RoboDK station: Example 1.1 - Linear rail & 2 fingers gripper Station.rdk

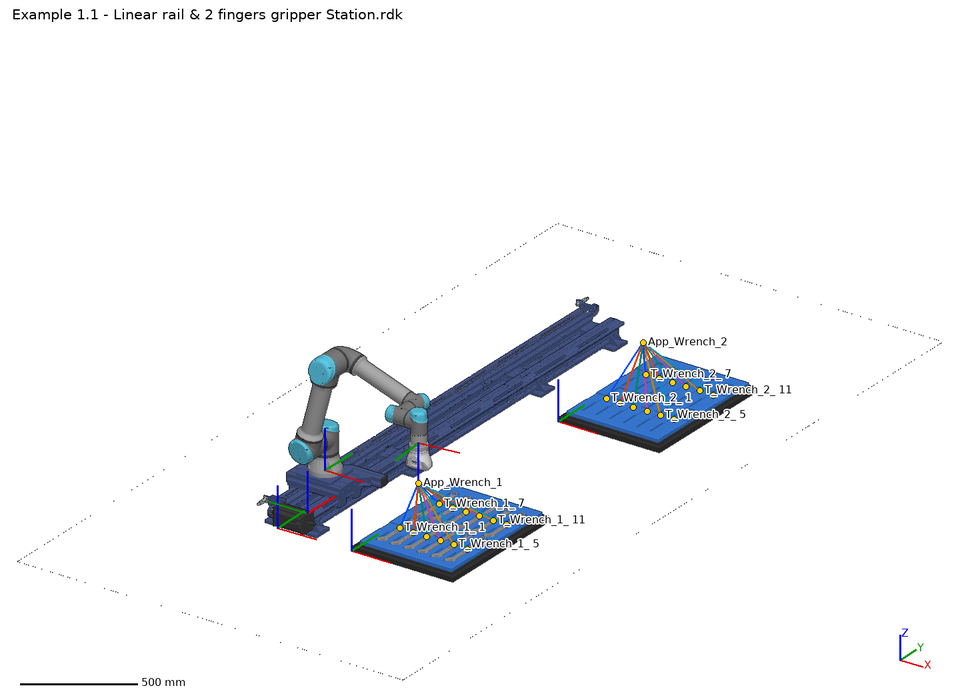
[picture v0: the station drawn from its stored meshes, robots at their saved joint values, targets as dots, program paths as lines]
Station Example 1.1 - 2 fingers gripper Station. Poses are relative to the parent item; angles as X-Y-Z fixed-axis rotations.
  - frame World at (0, 0, 0) mm
    - object Floor at (280, 1100, 0) mm, size 2000 x 4000 x 1 mm, geometry from plane_1m.sld
  - frame Linear Rail Base at (148.81, 12.71, 105) mm, rotated rx 0 ry 0 rz 90 deg
    - robot Linear Rail: 1 axes
        modified DH rows (alpha deg, a mm, theta deg, d mm): 0, 0, 0, 0 linear
        base shift (0, 0, 0) mm, rotated rx 0 ry 90 rz 0 deg
        joint limits [0] to [2100]; home [0]; saved at [150]
      - frame UR5e Base at (100, 85, 80) mm, rotated rx 0 ry 0 rz -90 deg
        - robot UR5e: 6 axes, payload 5 kg, reach 850 mm, repeatability 0.03 mm, weight 18.4 kg
            modified DH rows (alpha deg, a mm, theta deg, d mm): 0, 0, 0, 162.5; 90, 0, 180, 0; 0, 425, 0, 0; 0, 392.25, 0, 133.3; -90, 0, 0, 99.7; 90, 0, 180, 99.6
            joint limits [-360, -360, -360, -360, -360, -360] to [360, 360, 360, 360, 360, 360]; home [0, -90, -90, 0, 90, 0]; saved at [0, -104.57, -94.67, -70.76, 90, -95.16]
          - frame Schunk_Gripper Base at (0, 0, 0) mm
            - robot Schunk_Gripper: 1 axes
                joint limits [0] to [40]; home [40]; saved at [9]
            - target Gripper_Open (joint target) at (-117.49, 235.59, 143.86) mm; joints [40, 0, 0, 0, 0, 0] of Schunk_Gripper
            - target Gripper_Pick (joint target) at (0, 0, 150) mm; joints [9, 0, 0, 0, 0, 0] of Schunk_Gripper
          - tool Shunck_TCP, TCP at (0, 0, 190) mm
    - target Rail_Pos1 (joint target) at (150, 0, 0) mm; joints [150, 0, 0, 0, 0, nan] of Linear Rail
    - target Rail_Pos2 (joint target) at (1814.34, 0, 0) mm; joints [1814.34, 0, 0, 0, 0, 0] of Linear Rail
  - frame Frame Wrench 1 at (386.44, -2.63, 0) mm
    - object Jig at (0, 0, 0) mm, size 525 x 720 x 30 mm, geometry from Jig.step
    - object Wrench Matrix at (25, 25, 10) mm, size 475 x 670 x 40 mm, geometry from Matrix.step
    - target T_Wrench_1_ 1 (Cartesian target) at (100, 215, 50) mm, rotated rx 180 ry 0 rz 0 deg; joints [11.458, -119.591, -136.449, -13.961, 90, -78.542] of UR5e
    - target T_Wrench_1_ 2 (Cartesian target) at (170, 215, 50) mm, rotated rx 180 ry 0 rz 0 deg; joints [9.78, -123.515, -125.176, -21.309, 90, -80.22] of UR5e
    - target T_Wrench_1_ 3 (Cartesian target) at (240, 215, 50) mm, rotated rx 180 ry 0 rz 0 deg; joints [8.536, -128.193, -113.428, -28.378, 90, -81.464] of UR5e
    - target T_Wrench_1_ 4 (Cartesian target) at (310, 215, 50) mm, rotated rx 180 ry 0 rz 0 deg; joints [7.575, -133.539, -100.921, -35.54, 90, -82.425] of UR5e
    - target T_Wrench_1_ 5 (Cartesian target) at (380, 215, 50) mm, rotated rx 180 ry 0 rz 0 deg; joints [6.809, -139.644, -87.232, -43.124, 90, -83.191] of UR5e
    - target T_Wrench_1_ 6 (Cartesian target) at (450, 215, 50) mm, rotated rx 180 ry 0 rz 0 deg; joints [6.185, -146.811, -71.606, -51.583, 90, -83.815] of UR5e
    - target T_Wrench_1_ 7 (Cartesian target) at (100, 505, 50) mm, rotated rx 180 ry 0 rz 0 deg; joints [45.48, -122.94, -126.711, -20.349, 90, -44.52] of UR5e
    - target T_Wrench_1_ 8 (Cartesian target) at (170, 505, 50) mm, rotated rx 180 ry 0 rz 0 deg; joints [40.025, -126.988, -116.359, -26.653, 90, -49.975] of UR5e
    - target T_Wrench_1_ 9 (Cartesian target) at (240, 505, 50) mm, rotated rx 180 ry 0 rz 0 deg; joints [35.662, -131.694, -105.165, -33.141, 90, -54.338] of UR5e
    - target T_Wrench_1_ 10 (Cartesian target) at (310, 505, 50) mm, rotated rx 180 ry 0 rz 0 deg; joints [32.112, -137.097, -92.887, -40.015, 90, -57.888] of UR5e
    - target T_Wrench_1_ 11 (Cartesian target) at (380, 505, 50) mm, rotated rx 180 ry 0 rz 0 deg; joints [29.178, -143.374, -79.056, -47.57, 90, -60.822] of UR5e
    - target T_Wrench_1_ 12 (Cartesian target) at (450, 505, 50) mm, rotated rx 180 ry 0 rz 0 deg; joints [26.718, -150.974, -62.667, -56.359, 90, -63.282] of UR5e
    - target App_Wrench_1 (joint target) at (254.33, 132.05, 339.98) mm, rotated rx 180 ry 0 rz 5.16 deg; joints [0, -104.57, -94.67, -70.76, 90, -95.16] of UR5e
    - object Wrench 11 at (380, 505, 65) mm, size 44.5 x 267.3 x 18.4 mm, geometry from Wrench.step
    - object Wrench 12 at (450, 505, 65) mm, size 44.5 x 267.3 x 18.4 mm, geometry from Wrench.step
    - object Wrench 1 at (100, 215, 65) mm, size 44.5 x 267.3 x 18.4 mm, geometry from Wrench.step
    - object Wrench 2 at (170, 215, 65) mm, size 44.5 x 267.3 x 18.4 mm, geometry from Wrench.step
    - object Wrench 3 at (240, 215, 65) mm, size 44.5 x 267.3 x 18.4 mm, geometry from Wrench.step
    - object Wrench 4 at (310, 215, 65) mm, size 44.5 x 267.3 x 18.4 mm, geometry from Wrench.step
    - object Wrench 5 at (380, 215, 65) mm, size 44.5 x 267.3 x 18.4 mm, geometry from Wrench.step
    - object Wrench 6 at (450, 215, 65) mm, size 44.5 x 267.3 x 18.4 mm, geometry from Wrench.step
    - object Wrench 7 at (100, 505, 65) mm, size 44.5 x 267.3 x 18.4 mm, geometry from Wrench.step
    - object Wrench 8 at (170, 505, 65) mm, size 44.5 x 267.3 x 18.4 mm, geometry from Wrench.step
    - object Wrench 9 at (240, 505, 65) mm, size 44.5 x 267.3 x 18.4 mm, geometry from Wrench.step
    - object Wrench 10 at (310, 505, 65) mm, size 44.5 x 267.3 x 18.4 mm, geometry from Wrench.step
  - frame Frame Wrench 2 at (386.44, 1527.37, 0) mm
    - object Jig at (0, 0, 0) mm, size 525 x 720 x 30 mm, geometry from Jig.step
    - object Wrench Matrix at (25, 25, 10) mm, size 475 x 670 x 40 mm, geometry from Matrix.step
    - target T_Wrench_2_ 1 (Cartesian target) at (100, 215, 50) mm, rotated rx 180 ry 0 rz 0 deg; joints [11.458, -119.591, -136.449, -13.961, 90, -78.542] of UR5e
    - target T_Wrench_2_ 2 (Cartesian target) at (170, 215, 50) mm, rotated rx 180 ry 0 rz 0 deg; joints [9.78, -123.515, -125.176, -21.309, 90, -80.22] of UR5e
    - target T_Wrench_2_ 3 (Cartesian target) at (240, 215, 50) mm, rotated rx 180 ry 0 rz 0 deg; joints [8.536, -128.193, -113.428, -28.378, 90, -81.464] of UR5e
    - target T_Wrench_2_ 4 (Cartesian target) at (310, 215, 50) mm, rotated rx 180 ry 0 rz 0 deg; joints [7.575, -133.539, -100.921, -35.54, 90, -82.425] of UR5e
    - target T_Wrench_2_ 5 (Cartesian target) at (380, 215, 50) mm, rotated rx 180 ry 0 rz 0 deg; joints [6.809, -139.644, -87.232, -43.124, 90, -83.191] of UR5e
    - target T_Wrench_2_ 6 (Cartesian target) at (450, 215, 50) mm, rotated rx 180 ry 0 rz 0 deg; joints [6.185, -146.811, -71.606, -51.583, 90, -83.815] of UR5e
    - target T_Wrench_2_ 7 (Cartesian target) at (100, 505, 50) mm, rotated rx 180 ry 0 rz 0 deg; joints [45.48, -122.94, -126.711, -20.349, 90, -44.52] of UR5e
    - target T_Wrench_2_ 8 (Cartesian target) at (170, 505, 50) mm, rotated rx 180 ry 0 rz 0 deg; joints [40.025, -126.988, -116.359, -26.653, 90, -49.975] of UR5e
    - target T_Wrench_2_ 9 (Cartesian target) at (240, 505, 50) mm, rotated rx 180 ry 0 rz 0 deg; joints [35.662, -131.694, -105.165, -33.141, 90, -54.338] of UR5e
    - target T_Wrench_2_ 10 (Cartesian target) at (310, 505, 50) mm, rotated rx 180 ry 0 rz 0 deg; joints [32.112, -137.097, -92.887, -40.015, 90, -57.888] of UR5e
    - target T_Wrench_2_ 11 (Cartesian target) at (380, 505, 50) mm, rotated rx 180 ry 0 rz 0 deg; joints [29.178, -143.374, -79.056, -47.57, 90, -60.822] of UR5e
    - target T_Wrench_2_ 12 (Cartesian target) at (450, 505, 50) mm, rotated rx 180 ry 0 rz 0 deg; joints [26.718, -150.974, -62.667, -56.359, 90, -63.282] of UR5e
    - target App_Wrench_2 (joint target) at (254.33, 266.39, 339.98) mm, rotated rx 180 ry 0 rz 5.16 deg; joints [0, -104.57, -94.67, -70.76, 90, -95.16] of UR5e
  - program ReplaceObjects (1 instructions, listed below)
  - folder RailPositions
    - program RailPos1 (1 instructions, listed below)
    - program RailPos2 (1 instructions, listed below)
  - folder GripperPositions
    - program GripperPosPick (1 instructions, listed below)
    - program GripperPosOpen (1 instructions, listed below)
  - folder PickPrograms
    - program PickWrench (2 instructions, listed below)
    - program PickWrenchPos1 (6 instructions, listed below)
    - program PickWrenchPos2 (6 instructions, listed below)
    - program PickWrenchPos3 (6 instructions, listed below)
    - program PickWrenchPos4 (6 instructions, listed below)
    - program PickWrenchPos5 (6 instructions, listed below)
    - program PickWrenchPos6 (6 instructions, listed below)
    - program PickWrenchPos7 (6 instructions, listed below)
    - program PickWrenchPos8 (6 instructions, listed below)
    - program PickWrenchPos9 (6 instructions, listed below)
    - program PickWrenchPos10 (6 instructions, listed below)
    - program PickWrenchPos11 (6 instructions, listed below)
    - program PickWrenchPos12 (6 instructions, listed below)
  - folder PlacePrograms
    - program PlaceWrench (2 instructions, listed below)
    - program PlaceWrenchPos1 (6 instructions, listed below)
    - program PlaceWrenchPos2 (6 instructions, listed below)
    - program PlaceWrenchPos3 (6 instructions, listed below)
    - program PlaceWrenchPos4 (6 instructions, listed below)
    - program PlaceWrenchPos5 (6 instructions, listed below)
    - program PlaceWrenchPos6 (6 instructions, listed below)
    - program PlaceWrenchPos7 (6 instructions, listed below)
    - program PlaceWrenchPos8 (6 instructions, listed below)
    - program PlaceWrenchPos9 (6 instructions, listed below)
    - program PlaceWrenchPos10 (6 instructions, listed below)
    - program PlaceWrenchPos11 (6 instructions, listed below)
    - program PlaceWrenchPos12 (6 instructions, listed below)
  - program MainProgram (51 instructions, listed below)
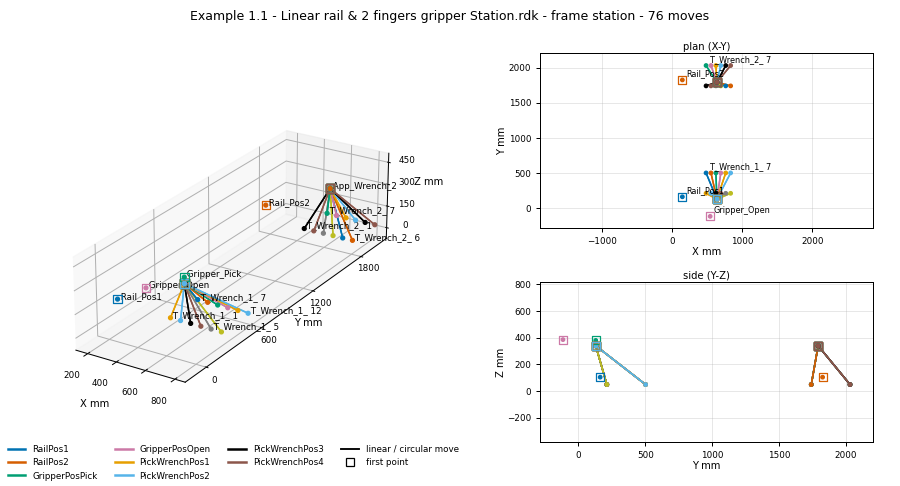
[picture p0: tool path of Example 1.1 - Linear rail & 2 fingers gripper Station.rdk in frame station, 76 of 76 moves have a stored position in this frame; points joined in program order, loops and branches not executed]

--- program ReplaceObjects (robot UR5e) ---
  Replace objects

--- program RailPos1 (robot Linear Rail) ---
  MoveJ (Rail_Pos1)

--- program RailPos2 (robot Linear Rail) ---
  MoveJ (Rail_Pos2)

--- program GripperPosPick (robot Schunk_Gripper) ---
  MoveJ (Gripper_Pick)

--- program GripperPosOpen (robot Schunk_Gripper) ---
  MoveJ (Gripper_Open)

--- program PickWrench (robot UR5e) ---
  Call GripperPosPick
  Attach to Shunck_TCP

--- program PickWrenchPos1 (robot UR5e) ---
  Set Ref.: Frame Wrench 1
  Set Tool: Shunck_TCP
  MoveJ (App_Wrench_1)
  MoveL (T_Wrench_1_ 1)
  Call PickWrench
  MoveL (App_Wrench_1)

--- program PickWrenchPos2 (robot UR5e) ---
  Set Ref.: Frame Wrench 1
  Set Tool: Shunck_TCP
  MoveJ (App_Wrench_1)
  MoveL (T_Wrench_1_ 2)
  Call PickWrench
  MoveL (App_Wrench_1)

--- program PickWrenchPos3 (robot UR5e) ---
  Set Ref.: Frame Wrench 1
  Set Tool: Shunck_TCP
  MoveJ (App_Wrench_1)
  MoveL (T_Wrench_1_ 3)
  Call PickWrench
  MoveL (App_Wrench_1)

--- program PickWrenchPos4 (robot UR5e) ---
  Set Ref.: Frame Wrench 1
  Set Tool: Shunck_TCP
  MoveJ (App_Wrench_1)
  MoveL (T_Wrench_1_ 4)
  Call PickWrench
  MoveL (App_Wrench_1)

--- program PickWrenchPos5 (robot UR5e) ---
  Set Ref.: Frame Wrench 1
  Set Tool: Shunck_TCP
  MoveJ (App_Wrench_1)
  MoveL (T_Wrench_1_ 5)
  Call PickWrench
  MoveL (App_Wrench_1)

--- program PickWrenchPos6 (robot UR5e) ---
  Set Ref.: Frame Wrench 1
  Set Tool: Shunck_TCP
  MoveJ (App_Wrench_1)
  MoveL (T_Wrench_1_ 6)
  Call PickWrench
  MoveL (App_Wrench_1)

--- program PickWrenchPos7 (robot UR5e) ---
  Set Ref.: Frame Wrench 1
  Set Tool: Shunck_TCP
  MoveJ (App_Wrench_1)
  MoveL (T_Wrench_1_ 7)
  Call PickWrench
  MoveL (App_Wrench_1)

--- program PickWrenchPos8 (robot UR5e) ---
  Set Ref.: Frame Wrench 1
  Set Tool: Shunck_TCP
  MoveJ (App_Wrench_1)
  MoveL (T_Wrench_1_ 8)
  Call PickWrench
  MoveL (App_Wrench_1)

--- program PickWrenchPos9 (robot UR5e) ---
  Set Ref.: Frame Wrench 1
  Set Tool: Shunck_TCP
  MoveJ (App_Wrench_1)
  MoveL (T_Wrench_1_ 9)
  Call PickWrench
  MoveL (App_Wrench_1)

--- program PickWrenchPos10 (robot UR5e) ---
  Set Ref.: Frame Wrench 1
  Set Tool: Shunck_TCP
  MoveJ (App_Wrench_1)
  MoveL (T_Wrench_1_ 10)
  Call PickWrench
  MoveL (App_Wrench_1)

--- program PickWrenchPos11 (robot UR5e) ---
  Set Ref.: Frame Wrench 1
  Set Tool: Shunck_TCP
  MoveJ (App_Wrench_1)
  MoveL (T_Wrench_1_ 11)
  Call PickWrench
  MoveL (App_Wrench_1)

--- program PickWrenchPos12 (robot UR5e) ---
  Set Ref.: Frame Wrench 1
  Set Tool: Shunck_TCP
  MoveJ (App_Wrench_1)
  MoveL (T_Wrench_1_ 12)
  Call PickWrench
  MoveL (App_Wrench_1)

--- program PlaceWrench (robot UR5e) ---
  Call GripperPosOpen
  Detach from Shunck_TCP

--- program PlaceWrenchPos1 (robot UR5e) ---
  Set Ref.: Frame Wrench 2
  Set Tool: Shunck_TCP
  MoveJ (App_Wrench_2)
  MoveL (T_Wrench_2_ 1)
  Call PlaceWrench
  MoveL (App_Wrench_2)

--- program PlaceWrenchPos2 (robot UR5e) ---
  Set Ref.: Frame Wrench 2
  Set Tool: Shunck_TCP
  MoveJ (App_Wrench_2)
  MoveL (T_Wrench_2_ 2)
  Call PlaceWrench
  MoveL (App_Wrench_2)

--- program PlaceWrenchPos3 (robot UR5e) ---
  Set Ref.: Frame Wrench 2
  Set Tool: Shunck_TCP
  MoveJ (App_Wrench_2)
  MoveL (T_Wrench_2_ 3)
  Call PlaceWrench
  MoveL (App_Wrench_2)

--- program PlaceWrenchPos4 (robot UR5e) ---
  Set Ref.: Frame Wrench 2
  Set Tool: Shunck_TCP
  MoveJ (App_Wrench_2)
  MoveL (T_Wrench_2_ 4)
  Call PlaceWrench
  MoveL (App_Wrench_2)

--- program PlaceWrenchPos5 (robot UR5e) ---
  Set Ref.: Frame Wrench 2
  Set Tool: Shunck_TCP
  MoveJ (App_Wrench_2)
  MoveL (T_Wrench_2_ 5)
  Call PlaceWrench
  MoveL (App_Wrench_2)

--- program PlaceWrenchPos6 (robot UR5e) ---
  Set Ref.: Frame Wrench 2
  Set Tool: Shunck_TCP
  MoveJ (App_Wrench_2)
  MoveL (T_Wrench_2_ 6)
  Call PlaceWrench
  MoveL (App_Wrench_2)

--- program PlaceWrenchPos7 (robot UR5e) ---
  Set Ref.: Frame Wrench 2
  Set Tool: Shunck_TCP
  MoveJ (App_Wrench_2)
  MoveL (T_Wrench_2_ 7)
  Call PlaceWrench
  MoveL (App_Wrench_2)

--- program PlaceWrenchPos8 (robot UR5e) ---
  Set Ref.: Frame Wrench 2
  Set Tool: Shunck_TCP
  MoveJ (App_Wrench_2)
  MoveL (T_Wrench_2_ 8)
  Call PlaceWrench
  MoveL (App_Wrench_2)

--- program PlaceWrenchPos9 (robot UR5e) ---
  Set Ref.: Frame Wrench 2
  Set Tool: Shunck_TCP
  MoveJ (App_Wrench_2)
  MoveL (T_Wrench_2_ 9)
  Call PlaceWrench
  MoveL (App_Wrench_2)

--- program PlaceWrenchPos10 (robot UR5e) ---
  Set Ref.: Frame Wrench 2
  Set Tool: Shunck_TCP
  MoveJ (App_Wrench_2)
  MoveL (T_Wrench_2_ 10)
  Call PlaceWrench
  MoveL (App_Wrench_2)

--- program PlaceWrenchPos11 (robot UR5e) ---
  Set Ref.: Frame Wrench 2
  Set Tool: Shunck_TCP
  MoveJ (App_Wrench_2)
  MoveL (T_Wrench_2_ 11)
  Call PlaceWrench
  MoveL (App_Wrench_2)

--- program PlaceWrenchPos12 (robot UR5e) ---
  Set Ref.: Frame Wrench 2
  Set Tool: Shunck_TCP
  MoveJ (App_Wrench_2)
  MoveL (T_Wrench_2_ 12)
  Call PlaceWrench
  MoveL (App_Wrench_2)

--- program MainProgram (robot UR5e) ---
  Call ReplaceObjects
  Call GripperPosOpen
  Call RailPos1
  Call PickWrenchPos1
  Call RailPos2
  Call PlaceWrenchPos1
  Call RailPos1
  Call PickWrenchPos2
  Call RailPos2
  Call PlaceWrenchPos2
  Call RailPos1
  Call PickWrenchPos3
  Call RailPos2
  Call PlaceWrenchPos3
  Call RailPos1
  Call PickWrenchPos4
  Call RailPos2
  Call PlaceWrenchPos4
  Call RailPos1
  Call PickWrenchPos5
  Call RailPos2
  Call PlaceWrenchPos5
  Call RailPos1
  Call PickWrenchPos6
  Call RailPos2
  Call PlaceWrenchPos6
  Call RailPos1
  Call PickWrenchPos7
  Call RailPos2
  Call PlaceWrenchPos7
  Call RailPos1
  Call PickWrenchPos8
  Call RailPos2
  Call PlaceWrenchPos8
  Call RailPos1
  Call PickWrenchPos9
  Call RailPos2
  Call PlaceWrenchPos9
  Call RailPos1
  Call PickWrenchPos10
  Call RailPos2
  Call PlaceWrenchPos10
  Call RailPos1
  Call PickWrenchPos11
  Call RailPos2
  Call PlaceWrenchPos11
  Call RailPos1
  Call PickWrenchPos12
  Call RailPos2
  Call PlaceWrenchPos12
  Call RailPos1
